PROGRAM POU_ProcesoEntrada
VAR
	PusherAzul: FB_Pusher;
	PusherVerde: FB_Pusher;
	PusherMetal: FB_Pusher;
END_VAR

(*Este POU se encarga de controlar la parte inicial del proceso, donde se separan los materiales de 
entrada por tipo. Para ello, se activa el proceso con el botón principal (botón MARCHA) y comienzan 
a moverse las diferentes cintas, activando los pushers cuando la detección corresponda con el objeto 
deseado. Si el sensor visual detecta el objeto configurado en sus características, entonces se pasa 
a detectar el flanco de bajada del Diffuse Sensor, activando los pushers en el momento adecuado *)

// SECCIÓN AZUL
PusherAzul(
	SENSOR:= GVL_Sorting.bDiffuseSensorA, FRONTAL:= GVL_Sorting.sPusherA.PusherFrontLimit, 
	CAMARA:= GVL_Sorting.bVisionSensorA, PUSHER=> GVL_Sorting.sPusherA.Pusher);

// SECCIÓN VERDE
PusherVerde(
	SENSOR:= GVL_Sorting.bDiffuseSensorV, FRONTAL:= GVL_Sorting.sPusherV.PusherFrontLimit, 
	CAMARA:= GVL_Sorting.bVisionSensorV, PUSHER=> GVL_Sorting.sPusherV.Pusher);

// SECCIÓN METAL
PusherMetal(
	SENSOR:= GVL_Sorting.bDiffuseSensorM, FRONTAL:= GVL_Sorting.sPusherM.PusherFrontLimit, 
	CAMARA:= GVL_Sorting.bVisionSensorM, PUSHER=> GVL_Sorting.sPusherM.Pusher);

END_PROGRAM

(* stored: Version 1.1.0.1, ProductVersion 3.1.4024.12
   POU POU_ProcesoEntrada: Id {af995422-f2b4-4fc9-9e2b-ddf55a5fe502}, SpecialFunc None *)
